Yaskawa INFORM job: AAA.JBI

/JOB
//NAME AAA
//POS
///NPOS 2,0,0,0,0,0
C00000=5934,50336,-3321,22658,-48022,-28299
C00001=5934,52719,-5061,23488,-45902,-28850
//INST
///DATE 2023/02/07 14:02
///ATTR SC,RW
///GROUP1 RB1
NOP
MOVL C00000 V=10.0 PL=8
MOVL C00001 V=10.0 PL=0
END
